# EPICS autosave request: support/ip/2-9/ipApp/Db/Omega_DP41_settings.req
$(P)$(R)ReadValues.SCAN
$(P)$(R)ReadSettingsScan.SCAN
$(P)$(R)SP1_Write.A
$(P)$(R)SP2_Write.A
$(P)$(R)SP3_Write.A
$(P)$(R)SP4_Write.A
